{attribute 'linkalways'} 
{attribute 'no_explicit_call' := 'This FB is a CLASS and must be accessed using methods or properties'}
{attribute 'enable_dynamic_creation'}
FUNCTION_BLOCK FINAL Node_LEFT EXTENDS Node
VAR
	str : _STRING('');
	size : _INT(0);
	out : _STRING('');
END_VAR

METHOD PUBLIC  Clone : I_Node
VAR
	pNode : POINTER TO Node_LEFT;
END_VAR
pNode := __NEW(Node_LEFT);
Clone := pNode^;
END_METHOD

METHOD FB_init : BOOL
VAR_INPUT
	bInitRetains : BOOL; // if TRUE, the retain variables are initialized (warm start / cold start)
	bInCopyCode : BOOL;  // if TRUE, the instance afterwards gets moved into the copy code (online change)
END_VAR
AddParameter('str', str);
AddParameter('size', size);
AddOutput('out', out);
END_METHOD

METHOD PROTECTED OnExecute
VAR
END_VAR
out.Value := LEFT(str.Value, size.Value);
END_METHOD

END_FUNCTION_BLOCK

(* stored: Version 1.1.0.1, ProductVersion 3.1.4026.18
   POU Node_LEFT: Id {2aff3026-7ee5-0755-15fe-b4758071897f}, SpecialFunc None
   Folder Constructor: Id {99dabb16-e669-0dad-0d46-622ddcd48dff}
   Method Clone: Id {67b60cd5-5b0d-0219-037c-d9ef1e9ee7e1}
   Method FB_init: Id {561507e3-3c52-02a1-3ae7-24a72b017606}
   Method OnExecute: Id {7aab1ebc-4a7b-0b74-3807-5eab05c0a030} *)
